FUNCTION_BLOCK FB_Brake_oil_pump
VAR_INPUT
	Run_cmd:BOOL;
	Stop_cmd:BOOL;
	Bop1_switch:BOOL;
	Bop1_tripped:BOOL;
	Bop1_running:BOOL;
	Bop1_use_internal_es:BOOL;
	Bop1_ext_estop:BOOL;
	Bop2_switch:BOOL;
	Bop2_tripped:BOOL;
	Bop2_running:BOOL;
	Bop2_use_internal_es:BOOL;
	Bop2_ext_estop:BOOL;
	Bop1_interlock:BOOL;
	Bop2_interlock:BOOL;
	Common_interlock:BOOL;
	Bridge1:BOOL;
	Bridge2:BOOL;
	Bridge3:BOOL;
	Pause_time:TIME;
	Reset:BOOL;
	Duty_bop1:REAL;
	Duty_bop2:REAL;
	Bop1_Reg455:REAL;
	Bop2_Reg455:REAL;
END_VAR
VAR_OUTPUT
	Bop1_run:BOOL;
	Bop2_run:BOOL;
	Bop1_ns_trip:BOOL;
	Bop1_es_trip:BOOL;
	Bop1_contactor_stuck:BOOL;
	Bop2_ns_trip:BOOL;
	Bop2_es_trip:BOOL;
	Bop2_contactor_stuck:BOOL;
	Start_output:BOOL;
	Bop1_Reg704:REAL;
	Bop1_Reg703:REAL;
	Bop1_Avg_curr:REAL;
	Bop2_Reg704:REAL;
	Bop2_Reg703:REAL;
	Bop2_Avg_curr:REAL;
END_VAR
VAR_IN_OUT
	Bop1_data:dut_Dol_Starter;
	Bop2_data:dut_Dol_Starter;
END_VAR
VAR
	FB_Duty_0: FB_Duty;
	FB_DOL_Control_0: FB_DOL_Control;
	FB_DOL_Control_1: FB_DOL_Control;
END_VAR

Brake_oil_pump();

METHOD Brake_oil_pump
VAR_INPUT
END_VAR
VAR_INST // added by the converter: edge detectors and wires of the graphical bodies
    _w1 : BOOL;
END_VAR
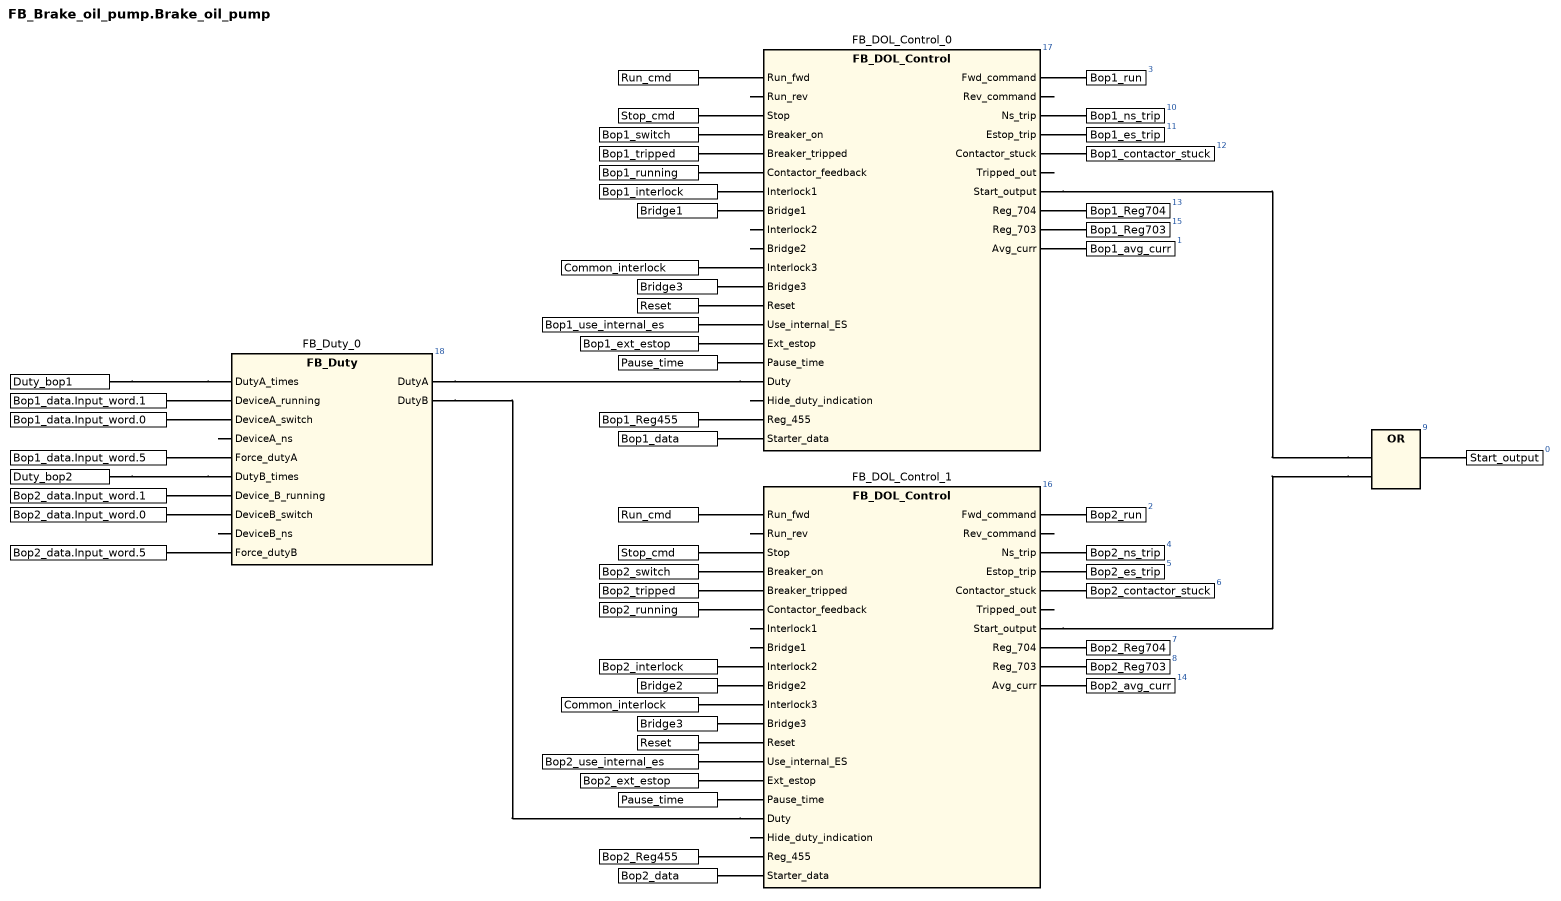
Start_output := _w1;
Bop1_avg_curr := FB_DOL_Control_0.Avg_curr;
Bop2_run := FB_DOL_Control_1.Fwd_command;
Bop1_run := FB_DOL_Control_0.Fwd_command;
Bop2_ns_trip := FB_DOL_Control_1.Ns_trip;
Bop2_es_trip := FB_DOL_Control_1.Estop_trip;
Bop2_contactor_stuck := FB_DOL_Control_1.Contactor_stuck;
Bop2_Reg704 := FB_DOL_Control_1.Reg_704;
Bop2_Reg703 := FB_DOL_Control_1.Reg_703;
_w1 := FB_DOL_Control_0.Start_output OR FB_DOL_Control_1.Start_output;
Bop1_ns_trip := FB_DOL_Control_0.Ns_trip;
Bop1_es_trip := FB_DOL_Control_0.Estop_trip;
Bop1_contactor_stuck := FB_DOL_Control_0.Contactor_stuck;
Bop1_Reg704 := FB_DOL_Control_0.Reg_704;
Bop2_avg_curr := FB_DOL_Control_1.Avg_curr;
Bop1_Reg703 := FB_DOL_Control_0.Reg_703;
FB_DOL_Control_1(
    Run_fwd := Run_cmd,
    Stop := Stop_cmd,
    Breaker_on := Bop2_switch,
    Breaker_tripped := Bop2_tripped,
    Contactor_feedback := Bop2_running,
    Interlock2 := Bop2_interlock,
    Bridge2 := Bridge2,
    Interlock3 := Common_interlock,
    Bridge3 := Bridge3,
    Reset := Reset,
    Use_internal_ES := Bop2_use_internal_es,
    Ext_estop := Bop2_ext_estop,
    Pause_time := Pause_time,
    Duty := FB_Duty_0.DutyB,
    Reg_455 := Bop2_Reg455,
    Starter_data := Bop2_data); // FB_DOL_Control
FB_DOL_Control_0(
    Run_fwd := Run_cmd,
    Stop := Stop_cmd,
    Breaker_on := Bop1_switch,
    Breaker_tripped := Bop1_tripped,
    Contactor_feedback := Bop1_running,
    Interlock1 := Bop1_interlock,
    Bridge1 := Bridge1,
    Interlock3 := Common_interlock,
    Bridge3 := Bridge3,
    Reset := Reset,
    Use_internal_ES := Bop1_use_internal_es,
    Ext_estop := Bop1_ext_estop,
    Pause_time := Pause_time,
    Duty := FB_Duty_0.DutyA,
    Reg_455 := Bop1_Reg455,
    Starter_data := Bop1_data); // FB_DOL_Control
FB_Duty_0(
    DutyA_times := Duty_bop1,
    DeviceA_running := Bop1_data.Input_word.1,
    DeviceA_switch := Bop1_data.Input_word.0,
    Force_dutyA := Bop1_data.Input_word.5,
    DutyB_times := Duty_bop2,
    Device_B_running := Bop2_data.Input_word.1,
    DeviceB_switch := Bop2_data.Input_word.0,
    Force_dutyB := Bop2_data.Input_word.5); // FB_Duty
END_METHOD

END_FUNCTION_BLOCK

(* stored: Version 1.1.0.1, ProductVersion 3.1.4024.0
   POU FB_Brake_oil_pump: Id {d9719d8f-ebbd-413b-a586-b463899a0318}, SpecialFunc None
   Method Brake_oil_pump: Id {00820402-07fb-43f2-840a-20acfcbd2696} *)
